FUNCTION_BLOCK FB_ManipAxis
VAR_INPUT
	i_xHotPlug	:	BOOL;
END_VAR
VAR_OUTPUT
	q_asResult: ARRAY [1..20] OF STRING;
	q_xError	:	BOOL;
END_VAR
VAR_IN_OUT
	iq_ManipAxis	:	ST_ManipAxis;
END_VAR
VAR

	mcPower	:	MC_Power;
	mcReset	:	MC_Reset;
	mcMoveAbsolute : ARRAY[1..2] OF MC_MoveAbsolute;
	mcHalt	:	MC_Halt;
	mcSmoothMover	:	MC_SmoothMover;
	//Error Stuff
	indexResult: INT := 1;
	fbFormatString	:	FB_FormatString;
	
	xInitComplete	:	BOOL := FALSE;
	
	imcBlockIndex: INT;
	
	rtEnable : R_TRIG;
	ftEnable : F_TRIG;
	rtStop	:	R_TRIG;
	rtStart	:	R_TRIG;
	rReqAbsPosOld: REAL := 0;
	rReqAbsPosPrevious: REAL;
	iI: INT;
END_VAR

(* Manipulator Axis Function Block
Alex Wallace, 2016-8-8 

This block works by jumping between two absolute move blocks and buffering
the motion between them.
*)


rtEnable(CLK:=iq_ManipAxis.xEnable);
ftEnable(CLK:=iq_ManipAxis.xEnable);

//Update status
iq_ManipAxis.stAxis();

IF rtEnable.Q OR ftEnable.Q THEN
	xInitComplete := FALSE;
	iq_ManipAxis.eState := Init;
ELSIF xInitComplete THEN
	iq_ManipAxis.eState := MoveEnabled;
END_IF

//For EPICS, because the modbus map was made for 32 bit..
iq_ManipAxis.rActPos := LREAL_TO_REAL(iq_ManipAxis.stAxis.NcToPlc.ActPos);


CASE iq_ManipAxis.eState OF
	0: iq_ManipAxis.eState := Init;
	Init:
	(* Start by initializing the motor axis *)
	mcPower.Enable := iq_ManipAxis.xEnable;
	iq_ManipAxis.rReqAbsPos := iq_ManipAxis.rActPos; //do this when the PLC comes up so we don't just lose the position if we tweak
	IF mcPower.Status THEN //success
		xInitComplete := TRUE;
		q_asResult[indexResult] := 'Motor init success';
		indexResult := indexResult + 1;
		iq_ManipAxis.eState := MoveEnabled;
	ELSIF mcPower.Error THEN
		mcPower.Enable := FALSE;
		fbFormatString(sFormat:='Init mcPower Error: %s', arg1:=F_UDINT(mcPower.ErrorID));
		ActError();
	END_IF
		
	MoveEnabled:
		mcSmoothMover.Enable := iq_ManipAxis.xEnable;
		mcSmoothMover.ReqAbsPos := LIMIT(-100, REAL_TO_LREAL(iq_ManipAxis.rReqAbsPos), 100);
		mcSmoothMover.Execute := iq_ManipAxis.xStart;
		(*We've already captured the rising edge of start (if there was one, so 
		go ahead and reset it.*)
		iq_ManipAxis.xStart := FALSE;
		
		//Halt
		mcHalt.Execute S= iq_ManipAxis.xStop;
		mcHalt.Execute R= mcHalt.Busy;
		iq_ManipAxis.xStop R= mcHalt.Busy;
		IF mcPower.Error OR mcSmoothMover.Error THEN
			iq_ManipAxis.eState:=Error;
		END_IF
	

	
END_CASE


mcReset.Execute := rtEnable.Q OR i_xHotPlug OR iq_ManipAxis.xReset;
//Reset the reset controls for the next reset
IF mcReset.Done THEN
	mcReset.Execute := FALSE;
	iq_ManipAxis.xReset := FALSE;
	iq_ManipAxis.eState:=Init;
END_IF
//Set function block state once axis is happy again
IF NOT iq_ManipAxis.stAxis.Status.Error THEN
	q_xError := FALSE;
END_IF


(* Run the mc blocks *)
ActPower();
mcReset(Axis:=iq_ManipAxis.stAxis);
mcSmoothMover(Axis:=iq_ManipAxis.stAxis,
	Velocity:=iq_ManipAxis.lrVelocity);
mcHalt(Axis:=iq_ManipAxis.stAxis);

iq_ManipAxis.xDmov := mcHalt.Done OR mcSmoothMover.Done;
iq_ManipAxis.xMovn := mcHalt.Busy OR mcSmoothMover.Busy;

//For display, this logic is not for safety
iq_ManipAxis.xHLS := NOT iq_ManipAxis.xHiLS;
iq_ManipAxis.xLLS := NOT iq_ManipAxis.xLoLS;

ACTION ActPower:
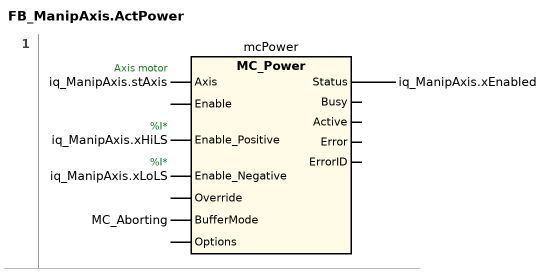
// NETWORK 1
//   iq_ManipAxis.stAxis: Axis motor
//   iq_ManipAxis.xHiLS: AT %I*
//   iq_ManipAxis.xLoLS: AT %I*
mcPower(
    Axis := iq_ManipAxis.stAxis,
    Enable_Positive := iq_ManipAxis.xHiLS,
    Enable_Negative := iq_ManipAxis.xLoLS,
    BufferMode := MC_Aborting); // MC_Power
iq_ManipAxis.xEnabled := mcPower.Status;
END_ACTION

ACTION ActError:
(* Error action
*)

//Reset the debugging index
IF indexResult > 20 THEN indexResult := 1; END_IF

iq_ManipAxis.eState := Error;
q_xError	:=	TRUE;
q_asResult[indexResult] := fbFormatString.sOut;
indexResult := indexResult +1;
END_ACTION

END_FUNCTION_BLOCK

(* stored: Version 1.1.0.1, ProductVersion 3.1.4020.12
   POU FB_ManipAxis: Id {2c576ec6-7433-4ec0-8547-ab9b5dd393c9}, SpecialFunc None
   Action ActPower: Id {31b74a81-1b68-4db8-b9a3-64793fff0f5a}
   Action ActError: Id {efb14a67-3fcd-4d5f-a82f-60b8d6779b53} *)
